// TIA Portal V21 export
DATA_BLOCK "CipTimer"   // DB637
{ S7_Optimized_Access := 'TRUE' }
// stored: AutoNumber false, MemoryReserve 100
   VAR
      Timer1 : IEC_TIMER;
      Timer2 { S7_SetPoint := 'True'} : IEC_TIMER;
      Timer3 { S7_SetPoint := 'True'} : IEC_TIMER;
      Timer4 { S7_SetPoint := 'True'} : IEC_TIMER;
      Timer5 { S7_SetPoint := 'True'} : IEC_TIMER;
   END_VAR
BEGIN
END_DATA_BLOCK
